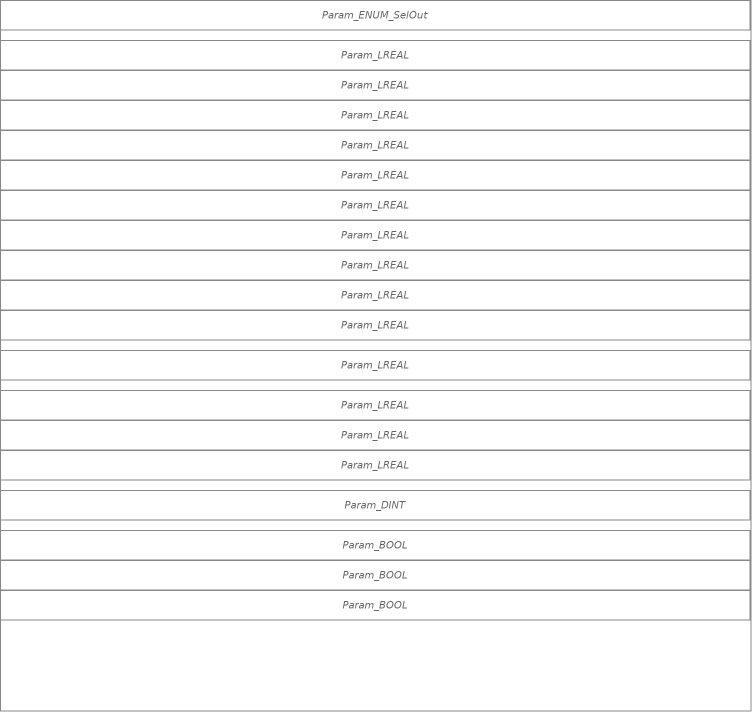
VISUALIZATION Visu_Mparam_Cool  // 752x712
    Frame (0,40 750x30)
        shows Param_LREAL(nIdx := 5)
    Frame (0,70 750x30)
        shows Param_LREAL(nIdx := 7)
    Frame (0,100 750x30)
        shows Param_LREAL(nIdx := 9)
    Frame (0,130 750x30)
        shows Param_LREAL(nIdx := 11)
    Frame (0,490 750x30)
        shows Param_DINT(nIdx := 10)
    Frame (0,0 750x30)
        shows Param_ENUM_SelOut(nIdx := 2)
    Frame (0,160 750x30)
        shows Param_LREAL(nIdx := 12)
    Frame (0,190 750x30)
        shows Param_LREAL(nIdx := 13)
    Frame (0,220 750x30)
        shows Param_LREAL(nIdx := 14)
    Frame (0,250 750x30)
        shows Param_LREAL(nIdx := 15)
    Frame (0,280 750x30)
        shows Param_LREAL(nIdx := 17)
    Frame (0,310 750x30)
        shows Param_LREAL(nIdx := 18)
    Frame (0,350 750x30)
        shows Param_LREAL(nIdx := 22)
    Frame (0,390 750x30)
        shows Param_LREAL(nIdx := 33)
    Frame (0,420 750x30)
        shows Param_LREAL(nIdx := 34)
    Frame (0,450 750x30)
        shows Param_LREAL(nIdx := 36)
    Frame (0,530 750x30)
        shows Param_BOOL(nIdx := 12)
    Frame (0,560 750x30)
        shows Param_BOOL(nIdx := 16)
    Frame (0,590 750x30)
        shows Param_BOOL(nIdx := 19)
    Rectangle (0,680 750x30)
END_VISUALIZATION

(* stored: Version 1.1.0.1, ProductVersion 3.1.4024.12
   Visu Visu_Mparam_Cool: Id {dd7220ea-a780-43a3-ab41-0e9437711069} *)
